Staubli VAL3: remGetHereSph.pgx

program remGetHereSph(string& sReturn[] (dimensions=1))
begin
  // Return current position in spherical coordinates.
  //
  logMsg("call remGetHere")
  call remCalcHereSph()
  sReturn="GETPOSSPH"
  sReturn=sReturn+" "+toString(sNumConv,nAzHere)
  sReturn=sReturn+" "+toString(sNumConv,nElHere)
  sReturn=sReturn+" "+toString(sNumConv,nRHere)
end
